// TIA Portal V18 export
// export: Created 2026-01-09T11:32:02.2991975Z, ExportSetting WithDefaults, DisplayName Totally Integrated Automation Portal, DisplayVersion V18 Update 5, DisplayName TIA Portal Openness, DisplayVersion V18 Update 5, DisplayName TIA Portal Teamcenter Gateway, DisplayVersion V18, DisplayName TIA Portal Version Control Interface, DisplayVersion V18, DisplayName SINAMICS Startdrive Advanced, DisplayVersion V18 SP2 Update 1, DisplayName SINAMICS Startdrive G110M, G120, G120C, G120D, G120P, G115D, DisplayVersion V18 SP2 Update 1, DisplayName SINAMICS Startdrive G130, G150, S120, S150, SINAMICS MV, S210, G220, S200, DisplayVersion V18 SP2 Update 1, DisplayName STEP 7 Professional, DisplayVersion V18 Update 5, DisplayName STEP 7 Safety, DisplayVersion V18, DisplayName WinCC Professional, DisplayVersion V18 Update 5
TagTable "P"
  DnstDataBlock_Profinet_Status{0} : Bool  (%DB[SysDDBNum].DBX132.0, CPU S71500-2PN_TP700, 1 s)
  DnstDataBlock_Profinet_Status{1} : Bool  (%DB[SysDDBNum].DBX132.1, CPU S71500-2PN_TP700, 1 s)
  DnstDataBlock_Profinet_Status{2} : Bool  (%DB[SysDDBNum].DBX132.2, CPU S71500-2PN_TP700, 1 s)
  DnstDataBlock_Profinet_Status{3} : Bool  (%DB[SysDDBNum].DBX132.3, CPU S71500-2PN_TP700, 1 s)
  DnstDataBlock_Profinet_Status{4} : Bool  (%DB[SysDDBNum].DBX132.4, CPU S71500-2PN_TP700, 1 s)
  DnstDataBlock_Profinet_Status{5} : Bool  (%DB[SysDDBNum].DBX132.5, CPU S71500-2PN_TP700, 1 s)
  DnstDataBlock_Profinet_Status{6} : Bool  (%DB[SysDDBNum].DBX132.6, CPU S71500-2PN_TP700, 1 s)
  DnstDataBlock_Profinet_Status{7} : Bool  (%DB[SysDDBNum].DBX132.7, CPU S71500-2PN_TP700, 1 s)
  DnstDataBlock_Profinet_Status{8} : Bool  (%DB[SysDDBNum].DBX133.0, CPU S71500-2PN_TP700, 1 s)
  DnstDataBlock_Profinet_Status{9} : Bool  (%DB[SysDDBNum].DBX133.1, CPU S71500-2PN_TP700, 1 s)
  DnstDataBlock_Profinet_Status{10} : Bool  (%DB[SysDDBNum].DBX133.2, CPU S71500-2PN_TP700, 1 s)
  DnstDataBlock_Profinet_Status{11} : Bool  (%DB[SysDDBNum].DBX133.3, CPU S71500-2PN_TP700, 1 s)
  DnstDataBlock_Profinet_Status{12} : Bool  (%DB[SysDDBNum].DBX133.4, CPU S71500-2PN_TP700, 1 s)
  DnstDataBlock_Profinet_Status{13} : Bool  (%DB[SysDDBNum].DBX133.5, CPU S71500-2PN_TP700, 1 s)
  DnstDataBlock_Profinet_Status{14} : Bool  (%DB[SysDDBNum].DBX133.6, CPU S71500-2PN_TP700, 1 s)
  DnstDataBlock_Profinet_Status{15} : Bool  (%DB[SysDDBNum].DBX133.7, CPU S71500-2PN_TP700, 1 s)
  DnstDataBlock_Profinet_Status{16} : Bool  (%DB[SysDDBNum].DBX134.0, CPU S71500-2PN_TP700, 1 s)
  DnstDataBlock_Profinet_Status{17} : Bool  (%DB[SysDDBNum].DBX134.1, CPU S71500-2PN_TP700, 1 s)
  DnstDataBlock_Profinet_Status{18} : Bool  (%DB[SysDDBNum].DBX134.2, CPU S71500-2PN_TP700, 1 s)
  DnstDataBlock_Profinet_Status{19} : Bool  (%DB[SysDDBNum].DBX134.3, CPU S71500-2PN_TP700, 1 s)
  DnstDataBlock_Profinet_Status{20} : Bool  (%DB[SysDDBNum].DBX134.4, CPU S71500-2PN_TP700, 1 s)
  DnstDataBlock_Profinet_Status{21} : Bool  (%DB[SysDDBNum].DBX134.5, CPU S71500-2PN_TP700, 1 s)
  DnstDataBlock_Profinet_Status{22} : Bool  (%DB[SysDDBNum].DBX134.6, CPU S71500-2PN_TP700, 1 s)
  DnstDataBlock_Profinet_Status{23} : Bool  (%DB[SysDDBNum].DBX134.7, CPU S71500-2PN_TP700, 1 s)
  DnstDataBlock_Profinet_Status{24} : Bool  (%DB[SysDDBNum].DBX135.0, CPU S71500-2PN_TP700, 1 s)
  DnstDataBlock_Profinet_Status{25} : Bool  (%DB[SysDDBNum].DBX135.1, CPU S71500-2PN_TP700, 1 s)
  DnstDataBlock_Profinet_Status{26} : Bool  (%DB[SysDDBNum].DBX135.2, CPU S71500-2PN_TP700, 1 s)
  DnstDataBlock_Profinet_Status{27} : Bool  (%DB[SysDDBNum].DBX135.3, CPU S71500-2PN_TP700, 1 s)
  DnstDataBlock_Profinet_Status{28} : Bool  (%DB[SysDDBNum].DBX135.4, CPU S71500-2PN_TP700, 1 s)
  DnstDataBlock_Profinet_Status{29} : Bool  (%DB[SysDDBNum].DBX135.5, CPU S71500-2PN_TP700, 1 s)
  DnstDataBlock_Profinet_Status{30} : Bool  (%DB[SysDDBNum].DBX135.6, CPU S71500-2PN_TP700, 1 s)
  DnstDataBlock_Profinet_Status{31} : Bool  (%DB[SysDDBNum].DBX135.7, CPU S71500-2PN_TP700, 1 s)
  DnstDataBlock_Profinet_Status{32} : Bool  (%DB[SysDDBNum].DBX136.0, CPU S71500-2PN_TP700, 1 s)
  DnstDataBlock_Profinet_Status{33} : Bool  (%DB[SysDDBNum].DBX136.1, CPU S71500-2PN_TP700, 1 s)
  DnstDataBlock_Profinet_Status{34} : Bool  (%DB[SysDDBNum].DBX136.2, CPU S71500-2PN_TP700, 1 s)
  DnstDataBlock_Profinet_Status{35} : Bool  (%DB[SysDDBNum].DBX136.3, CPU S71500-2PN_TP700, 1 s)
  DnstDataBlock_Profinet_Status{36} : Bool  (%DB[SysDDBNum].DBX136.4, CPU S71500-2PN_TP700, 1 s)
  DnstDataBlock_Profinet_Status{37} : Bool  (%DB[SysDDBNum].DBX136.5, CPU S71500-2PN_TP700, 1 s)
  DnstDataBlock_Profinet_Status{38} : Bool  (%DB[SysDDBNum].DBX136.6, CPU S71500-2PN_TP700, 1 s)
  DnstDataBlock_Profinet_Status{39} : Bool  (%DB[SysDDBNum].DBX136.7, CPU S71500-2PN_TP700, 1 s)
  DnstDataBlock_Profinet_Status{40} : Bool  (%DB[SysDDBNum].DBX137.0, CPU S71500-2PN_TP700, 1 s)
  DnstDataBlock_Profinet_Status{41} : Bool  (%DB[SysDDBNum].DBX137.1, CPU S71500-2PN_TP700, 1 s)
  DnstDataBlock_Profinet_Status{42} : Bool  (%DB[SysDDBNum].DBX137.2, CPU S71500-2PN_TP700, 1 s)
  DnstDataBlock_Profinet_Status{43} : Bool  (%DB[SysDDBNum].DBX137.3, CPU S71500-2PN_TP700, 1 s)
  DnstDataBlock_Profinet_Status{44} : Bool  (%DB[SysDDBNum].DBX137.4, CPU S71500-2PN_TP700, 1 s)
  DnstDataBlock_Profinet_Status{45} : Bool  (%DB[SysDDBNum].DBX137.5, CPU S71500-2PN_TP700, 1 s)
  DnstDataBlock_Profinet_Status{46} : Bool  (%DB[SysDDBNum].DBX137.6, CPU S71500-2PN_TP700, 1 s)
  DnstDataBlock_Profinet_Status{47} : Bool  (%DB[SysDDBNum].DBX137.7, CPU S71500-2PN_TP700, 1 s)
  DnstDataBlock_Profinet_Status{48} : Bool  (%DB[SysDDBNum].DBX138.0, CPU S71500-2PN_TP700, 1 s)
  DnstDataBlock_Profinet_Status{49} : Bool  (%DB[SysDDBNum].DBX138.1, CPU S71500-2PN_TP700, 1 s)
  DnstDataBlock_Profinet_Status{50} : Bool  (%DB[SysDDBNum].DBX138.2, CPU S71500-2PN_TP700, 1 s)
  DnstDataBlock_Profinet_Status{51} : Bool  (%DB[SysDDBNum].DBX138.3, CPU S71500-2PN_TP700, 1 s)
  DnstDataBlock_Profinet_Status{52} : Bool  (%DB[SysDDBNum].DBX138.4, CPU S71500-2PN_TP700, 1 s)
  DnstDataBlock_Profinet_Status{53} : Bool  (%DB[SysDDBNum].DBX138.5, CPU S71500-2PN_TP700, 1 s)
  DnstDataBlock_Profinet_Status{54} : Bool  (%DB[SysDDBNum].DBX138.6, CPU S71500-2PN_TP700, 1 s)
  DnstDataBlock_Profinet_Status{55} : Bool  (%DB[SysDDBNum].DBX138.7, CPU S71500-2PN_TP700, 1 s)
  DnstDataBlock_Profinet_Status{56} : Bool  (%DB[SysDDBNum].DBX139.0, CPU S71500-2PN_TP700, 1 s)
  DnstDataBlock_Profinet_Status{57} : Bool  (%DB[SysDDBNum].DBX139.1, CPU S71500-2PN_TP700, 1 s)
  DnstDataBlock_Profinet_Status{58} : Bool  (%DB[SysDDBNum].DBX139.2, CPU S71500-2PN_TP700, 1 s)
  DnstDataBlock_Profinet_Status{59} : Bool  (%DB[SysDDBNum].DBX139.3, CPU S71500-2PN_TP700, 1 s)
  DnstDataBlock_Profinet_Status{60} : Bool  (%DB[SysDDBNum].DBX139.4, CPU S71500-2PN_TP700, 1 s)
  DnstDataBlock_Profinet_Status{61} : Bool  (%DB[SysDDBNum].DBX139.5, CPU S71500-2PN_TP700, 1 s)
  DnstDataBlock_Profinet_Status{62} : Bool  (%DB[SysDDBNum].DBX139.6, CPU S71500-2PN_TP700, 1 s)
  DnstDataBlock_Profinet_Status{63} : Bool  (%DB[SysDDBNum].DBX139.7, CPU S71500-2PN_TP700, 1 s)
  DnstDataBlock_Profinet_Status{64} : Bool  (%DB[SysDDBNum].DBX140.0, CPU S71500-2PN_TP700, 1 s)
  DnstDataBlock_Profinet_Status{65} : Bool  (%DB[SysDDBNum].DBX140.1, CPU S71500-2PN_TP700, 1 s)
  DnstDataBlock_Profinet_Status{66} : Bool  (%DB[SysDDBNum].DBX140.2, CPU S71500-2PN_TP700, 1 s)
  DnstDataBlock_Profinet_Status{67} : Bool  (%DB[SysDDBNum].DBX140.3, CPU S71500-2PN_TP700, 1 s)
  DnstDataBlock_Profinet_Status{68} : Bool  (%DB[SysDDBNum].DBX140.4, CPU S71500-2PN_TP700, 1 s)
  DnstDataBlock_Profinet_Status{69} : Bool  (%DB[SysDDBNum].DBX140.5, CPU S71500-2PN_TP700, 1 s)
  DnstDataBlock_Profinet_Status{70} : Bool  (%DB[SysDDBNum].DBX140.6, CPU S71500-2PN_TP700, 1 s)
  DnstDataBlock_Profinet_Status{71} : Bool  (%DB[SysDDBNum].DBX140.7, CPU S71500-2PN_TP700, 1 s)
  DnstDataBlock_Profinet_Status{72} : Bool  (%DB[SysDDBNum].DBX141.0, CPU S71500-2PN_TP700, 1 s)
  DnstDataBlock_Profinet_Status{73} : Bool  (%DB[SysDDBNum].DBX141.1, CPU S71500-2PN_TP700, 1 s)
  DnstDataBlock_Profinet_Status{74} : Bool  (%DB[SysDDBNum].DBX141.2, CPU S71500-2PN_TP700, 1 s)
  DnstDataBlock_Profinet_Status{75} : Bool  (%DB[SysDDBNum].DBX141.3, CPU S71500-2PN_TP700, 1 s)
  DnstDataBlock_Profinet_Status{76} : Bool  (%DB[SysDDBNum].DBX141.4, CPU S71500-2PN_TP700, 1 s)
  DnstDataBlock_Profinet_Status{77} : Bool  (%DB[SysDDBNum].DBX141.5, CPU S71500-2PN_TP700, 1 s)
  DnstDataBlock_Profinet_Status{78} : Bool  (%DB[SysDDBNum].DBX141.6, CPU S71500-2PN_TP700, 1 s)
  DnstDataBlock_Profinet_Status{79} : Bool  (%DB[SysDDBNum].DBX141.7, CPU S71500-2PN_TP700, 1 s)
  DnstDataBlock_Profinet_Status{80} : Bool  (%DB[SysDDBNum].DBX142.0, CPU S71500-2PN_TP700, 1 s)
  DnstDataBlock_Profinet_Status{81} : Bool  (%DB[SysDDBNum].DBX142.1, CPU S71500-2PN_TP700, 1 s)
  DnstDataBlock_Profinet_Status{82} : Bool  (%DB[SysDDBNum].DBX142.2, CPU S71500-2PN_TP700, 1 s)
  DnstDataBlock_Profinet_Status{83} : Bool  (%DB[SysDDBNum].DBX142.3, CPU S71500-2PN_TP700, 1 s)
  DnstDataBlock_Profinet_Status{84} : Bool  (%DB[SysDDBNum].DBX142.4, CPU S71500-2PN_TP700, 1 s)
  DnstDataBlock_Profinet_Status{85} : Bool  (%DB[SysDDBNum].DBX142.5, CPU S71500-2PN_TP700, 1 s)
  DnstDataBlock_Profinet_Status{86} : Bool  (%DB[SysDDBNum].DBX142.6, CPU S71500-2PN_TP700, 1 s)
  DnstDataBlock_Profinet_Status{87} : Bool  (%DB[SysDDBNum].DBX142.7, CPU S71500-2PN_TP700, 1 s)
  DnstDataBlock_Profinet_Status{88} : Bool  (%DB[SysDDBNum].DBX143.0, CPU S71500-2PN_TP700, 1 s)
  DnstDataBlock_Profinet_Status{89} : Bool  (%DB[SysDDBNum].DBX143.1, CPU S71500-2PN_TP700, 1 s)
  DnstDataBlock_Profinet_Status{90} : Bool  (%DB[SysDDBNum].DBX143.2, CPU S71500-2PN_TP700, 1 s)
  DnstDataBlock_Profinet_Status{91} : Bool  (%DB[SysDDBNum].DBX143.3, CPU S71500-2PN_TP700, 1 s)
  DnstDataBlock_Profinet_Status{92} : Bool  (%DB[SysDDBNum].DBX143.4, CPU S71500-2PN_TP700, 1 s)
  DnstDataBlock_Profinet_Status{93} : Bool  (%DB[SysDDBNum].DBX143.5, CPU S71500-2PN_TP700, 1 s)
  DnstDataBlock_Profinet_Status{94} : Bool  (%DB[SysDDBNum].DBX143.6, CPU S71500-2PN_TP700, 1 s)
  DnstDataBlock_Profinet_Status{95} : Bool  (%DB[SysDDBNum].DBX143.7, CPU S71500-2PN_TP700, 1 s)
  DnstDataBlock_Profinet_Status{96} : Bool  (%DB[SysDDBNum].DBX144.0, CPU S71500-2PN_TP700, 1 s)
  DnstDataBlock_Profinet_Status{97} : Bool  (%DB[SysDDBNum].DBX144.1, CPU S71500-2PN_TP700, 1 s)
  DnstDataBlock_Profinet_Status{98} : Bool  (%DB[SysDDBNum].DBX144.2, CPU S71500-2PN_TP700, 1 s)
  DnstDataBlock_Profinet_Status{99} : Bool  (%DB[SysDDBNum].DBX144.3, CPU S71500-2PN_TP700, 1 s)
  DnstDataBlock_Profinet_Status{100} : Bool  (%DB[SysDDBNum].DBX144.4, CPU S71500-2PN_TP700, 1 s)
  DnstDataBlock_Profinet_Status{101} : Bool  (%DB[SysDDBNum].DBX144.5, CPU S71500-2PN_TP700, 1 s)
  DnstDataBlock.Profinet.Index : Word  (%DB[SysDDBNum].DBW130, CPU S71500-2PN_TP700, 1 s)
